PROGRAM MAIN
VAR
	fbMBWriteSingleReg :FB_MBWriteSingleReg ;
	nWriteValue : INT ;
	fbTrigger : R_TRIG ;
	eWriteState : (WAIT, TRIGGER, WRITE) ;
END_VAR

fbTrigger () ;
IF fbTrigger.Q THEN
	IF eReadState = WAIT THEN
		eReadState := Trigger ;
	END_IF
END_IF
CASE eReadState 
	WAIT:
	//bişey yazılmıyor.
	
	TRIGGER :
	FB_MBWriteSingleReg(
	sIPAddr:= '127.0.0.1', 
	nTCPPort:= 502, 
	nUnitID:= 16#FF, 
	nMBAddr:= , 
	nValue:= , 
	bExecute:= , 
	tTimeout:= , 
	bBusy=> , 
	bError=> , 
	nErrId=> );
END_CASE

END_PROGRAM

(* stored: Version 1.1.0.1, ProductVersion 3.1.4024.12
   POU MAIN: Id {a0d81122-dc44-41a3-b4f3-396835bb4bab}, SpecialFunc None *)
